TYPE stRawInput :
STRUCT
	Start	:	BOOL;
	Stop	:	BOOL;
	Emg		:	BOOL;
	Ack		:	BOOL;
	FC1		:	BOOL;
	FC2		:	BOOL;
END_STRUCT
END_TYPE

(* stored: Version 1.1.0.1
   DUT stRawInput: Id {2b5d9fb3-ffb1-0ce5-293f-82fcda668572} *)
